FUNCTION_BLOCK FB_VFCModbus1 IMPLEMENTS I_VolumeFlowController
VAR_INPUT CONSTANT
	fbModbusMaster	:	POINTER TO FB_TVRModbusMaster;
	nUnitID			:	BYTE;
END_VAR
VAR_OUTPUT
END_VAR
VAR
	//Properties
	bError 			: 	BOOL := FALSE;
	fNominalVolFlow	: 	REAL := 3690;
	fVolFlowSet 	: 	REAL := 0;
	fVolFlowAct		: 	REAL;
	
	bFinish 		:	BOOL;
	
END_VAR

PROPERTY Error : BOOL
GET
Error := THIS^.bError;
END_GET
SET
THIS^.bError := Error;
END_SET
END_PROPERTY

PROPERTY NominalVolumeFlow : REAL
GET
NominalVolumeFlow := THIS^.fNominalVolFlow;
END_GET
SET
THIS^.fNominalVolFlow := NominalVolumeFlow;
END_SET
END_PROPERTY

METHOD Run : BOOL
//Write properties to master
fbModbusMaster^.NominalVolumeFlow := fNominalVolFlow;
fbModbusMaster^.VolumeFlowSetpoint := fVolFlowSet;
fbModbusMaster^.UnitID := nUnitID;

//Execute modbus master
bFinish := fbModbusMaster^.Run();

//Read properties from master
bError := fbModbusMaster^.Error;
IF bFinish THEN
	fVolFlowAct := fbModbusMaster^.VolumeFlowActual;
END_IF

Run := bFinish;
END_METHOD

PROPERTY UnitID : BYTE
GET
UnitID := THIS^.nUnitID;
END_GET
SET
THIS^.nUnitID := UnitID;
END_SET
END_PROPERTY

PROPERTY VolumeFlowActual : REAL
GET
VolumeFlowActual := THIS^.fVolFlowAct;
END_GET
SET
THIS^.fVolFlowAct := VolumeFlowActual;
END_SET
END_PROPERTY

PROPERTY VolumeFlowSetpoint : REAL
GET
VolumeFlowSetpoint := THIS^.fVolFlowSet;
END_GET
SET
THIS^.fVolFlowSet := VolumeFlowSetpoint;
END_SET
END_PROPERTY

END_FUNCTION_BLOCK

(* stored: Version 1.1.0.1, ProductVersion 3.1.4024.0
   POU FB_VFCModbus1: Id {f74b13a1-24d8-459b-8dce-a8fe0c542ced}, SpecialFunc None
   Property Error: Id {71b9df27-f562-42dc-9fef-8d745f75ee2d}
   Get Get: Id {27f8f24d-e8ae-4570-b368-21f7d23d67ee}
   Set Set: Id {486ba3fa-cad5-475a-96ab-af6a993eb11c}
   Property NominalVolumeFlow: Id {d4d473d2-5010-4281-839e-81d451e3f3c4}
   Get Get: Id {0b8eb2d2-a948-42a2-a6fa-3a8ea967685c}
   Set Set: Id {eae288c3-362d-4a86-899f-d0e08424044e}
   Method Run: Id {994975af-7ebb-47ac-8340-8f7fb171efe0}
   Property UnitID: Id {294a349a-b4da-4c91-8d3f-c41c30e7520a}
   Get Get: Id {2e03ae53-8cbe-4b2a-8795-7d50765cb2a4}
   Set Set: Id {6c11174a-fb6c-4db9-b16d-7129ba1ffdf1}
   Property VolumeFlowActual: Id {a02d0020-e61c-45fd-b7e9-6e7640e87f19}
   Get Get: Id {45e73cc8-73d8-4999-b875-67ff53863fdf}
   Set Set: Id {df62dcfd-b20e-40da-a911-50cab1c2acd3}
   Property VolumeFlowSetpoint: Id {54411097-a2e4-47bc-8489-967168d417a1}
   Get Get: Id {93b02cf6-0ba3-4546-b983-345d2c2baefe}
   Set Set: Id {6374b22c-01ea-4d79-a793-bd4d1ad26b1f} *)
